(****************************************************************
NAME:			FB_SetPhaseUpperAxisPosition
DATA:			2022.10.18
VERSION:		1.0.0
DESCRIPTION:	FB_SetPhaseUpperAxisPosition
HISTORY:
				2022.10.18		NEW

***************************************************************)
FUNCTION_BLOCK FB_SetPhaseUpperAxisPosition
VAR_INPUT
	ValueSet:LREAL:=0;
	Execute:BOOL;
END_VAR
VAR_OUTPUT
	FbID:DINT:=1001;
	State:DINT;
	Busy:BOOL;
	Done:BOOL;
	Error:BOOL;
	ErrorID:DINT;
END_VAR
VAR
	PhaseUpperLin_MC_SetPosition: MC_SetPosition;
	fb_ton: TON;
	FB_PlcEmergencyStop: FB_PlcEmergencyStop;
END_VAR

IF Execute THEN
Busy:=TRUE;
Done:=FALSE;
fb_ton(PT:=t#0.1s);
CASE State OF
	0:
		IF PhaseUpperLin_MC_SetPosition.Error THEN		(*FB Error*)
			ErrorID:=1;
			State:=99;
		ELSE
			State:=1;
		END_IF
	1:	(*Execute*)
		PhaseUpperLin_MC_SetPosition.Position:=ValueSet;
		PhaseUpperLin_MC_SetPosition.Execute:=TRUE;
		A_SetPhaseUpperPositionMC();
		fb_ton.IN:=TRUE;
		State:=2;
	2:	(*Wait*)
		A_SetPhaseUpperPositionMC();
		IF NOT PhaseUpperLin_MC_SetPosition.Done THEN		
			IF NOT fb_ton.Q THEN
				State:=2;
			ELSE
				ErrorID:=4;
				State:=99;
			END_IF
		ELSIF  PhaseUpperLin_MC_SetPosition.Done THEN	
			State:=88;
		ELSE
			ErrorID:=5;
			State:=99;
		END_IF
	88:
		Execute:=FALSE;
		State:=0;
		Busy:=FALSE;
		Done:=TRUE;
		Error:=FALSE;
		ErrorID:=0;
		PhaseUpperLin_MC_SetPosition.Execute:=FALSE;
		fb_ton.IN:=FALSE;
	99:
		Execute:=FALSE;
		State:=99;
		Busy:=FALSE;
		Done:=FALSE;
		Error:=TRUE;
		PhaseUpperLin_MC_SetPosition.Execute:=FALSE;
		fb_ton.IN:=FALSE;
	-100:
		FB_PlcEmergencyStop();
		Execute:=FALSE;
		State:=-100;
		Busy:=FALSE;
		Done:=FALSE;
		Error:=TRUE;
		PhaseUpperLin_MC_SetPosition.Execute:=FALSE;
		fb_ton.IN:=FALSE;
END_CASE
END_IF

ACTION A_SetPhaseUpperPositionMC:
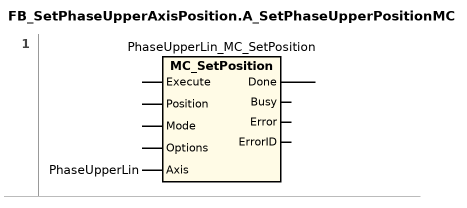
// NETWORK 1
PhaseUpperLin_MC_SetPosition(Axis := PhaseUpperLin); // MC_SetPosition
END_ACTION

END_FUNCTION_BLOCK

(* stored: Version 1.1.0.1, ProductVersion 3.1.4024.6
   POU FB_SetPhaseUpperAxisPosition: Id {9063ae89-4960-4401-841c-c79b07de8545}, SpecialFunc None
   Action A_SetPhaseUpperPositionMC: Id {362dde97-a54d-4198-8a53-3292d52617ea} *)
